(* CODESYS project tc3_mc3definitions.library
   TcLibraryId: Beckhoff Automation GmbH|Tc3_Mc3Definitions|3.2.38.0
   Company: Beckhoff Automation GmbH
   DefaultNamespace: Tc3_Mc3Definitions
   Version: 3.2.38.0
   Placeholder: Tc3_Mc3Definitions
   Title: Tc3_Mc3Definitions

Project tree, tasks and I/O mapping:
  Version/
    global variables Global_Version
  DUTs/
    Enums/
      data type MC_BUFFER_MODE
      data type MC_COMPENSATION_TYPE
      data type MC_DIRECTION
      data type MC_EXECUTION_MODE
      data type MC_SYNC_MODE
      data type MC_SYNC_STRATEGY
      data type MC_SYNC_DIRECTIONS
  GVLs/
    global variables GVL
*)

// DUTs/Enums/MC_BUFFER_MODE

(* Buffer mode between buffered commands. *)
	{attribute 'TcIecLibraryType'}
{attribute 'Namespace' := 'MC'}
TYPE MC_BUFFER_MODE : (mcAborting:=0, mcBuffered:=1, mcBlendingLow:=18, mcBlendingPrevious:=19, mcBlendingNext:=20, mcBlendingHigh:=21) UINT;
END_TYPE

// DUTs/Enums/MC_COMPENSATION_TYPE

(* Compensation type. *)
	{attribute 'TcIecLibraryType'}
{attribute 'Namespace' := 'MC'}
TYPE MC_COMPENSATION_TYPE : (mcTypeInvalidCompensation:=0, mcTypeGeoCompensation:=1) UINT;
END_TYPE

// DUTs/Enums/MC_DIRECTION

(* Defines the direction of the movement (e.g for an Modulo Axis). *)
	{attribute 'TcIecLibraryType'}
{attribute 'Namespace' := 'MC'}
TYPE MC_DIRECTION : (
	mcDirectionNonModulo:=0, 	(* Position is interpreted as absolute position. *)
	mcDirectionPositive:=1, 	(* Moves in positive direction. *)
	mcDirectionShortestWay:=2, 	(* The direction of movement depends on whether the positive direction of movement or the negative direction of movement is the shortest distance from the target position. *)
	mcDirectionNegative:=3	(* Moves in negative direction. *)
) UINT;
END_TYPE

// DUTs/Enums/MC_EXECUTION_MODE

(* Execution mode. *)
	{attribute 'TcIecLibraryType'}
{attribute 'Namespace' := 'MC'}
{attribute 'hide'}
TYPE MC_EXECUTION_MODE : (mcExecModeImmediately:=0, mcExecModeDelayed:=1, mcExecModeQueued:=2) UINT;
END_TYPE

// DUTs/Enums/MC_SYNC_MODE

(* Defines the direction of the synchronization position of modulo axes. *)
	{attribute 'TcIecLibraryType'}
{attribute 'Namespace' := 'MC'}
TYPE MC_SYNC_MODE : (
	mcSyncModeNonModulo:=0, 	(* SyncSlavePosition is interpreted as absolute position. *)
	mcSyncModePositive:=1, 	(* Synchronizes in positive direction. *)
	mcSyncModeNegative:=3	(* Synchronizes in negative direction. *)
) UINT;
END_TYPE

// DUTs/Enums/MC_SYNC_STRATEGY

(* Execution mode. *)
	{attribute 'TcIecLibraryType'}
{attribute 'Namespace' := 'MC'}
TYPE MC_SYNC_STRATEGY : (mcSyncStrategyLate:=1, mcSyncStrategySlow:=2, mcSyncStrategyEarly:=3) UINT;
END_TYPE

// DUTs/Enums/MC_SYNC_DIRECTIONS

(* Directions in which a slave is allowed to move during synchronizing phase. *)
	{attribute 'TcIecLibraryType'}
{attribute 'qualified_only'}
TYPE MC_SYNC_DIRECTIONS : (
		{attribute 'hide'}
Invalid:=0, 	(* Indicates invalid information, e.g. no connection or component not yet ready. *)
	Positive:=1, 	(* Movement is allowed only in positive direction while synchronizing. *)
	Negative:=2, 	(* Movement is allowed only in negative direction while synchronizing. *)
	Both:=3	(* Movement is allowed in any direction while synchronizing. *)
) UINT := Invalid;
END_TYPE

// Version/Global_Version
{attribute 'TcGenerated'}
// This function has been automatically generated from the project information.
VAR_GLOBAL CONSTANT
	{attribute 'const_non_replaced'}
	{attribute 'linkalways'}
	stLibVersion_Tc3_Mc3Definitions : ST_LibVersion := (iMajor := 3, iMinor := 2, iBuild := 38, iRevision := 0, sVersion := '3.2.38.0');
	{attribute 'const_non_replaced'}
	{attribute 'linkalways'}
	sLibraryId_Tc3_Mc3Definitions : String := 'Beckhoff Automation GmbH|Tc3_Mc3Definitions|3.2.38.0';
END_VAR

// GVLs/GVL

VAR_GLOBAL CONSTANT
		MC_DEFAULT	:	LREAL := 1E300;
		MC_IGNORE	:	LREAL := 1E301;
		MC_INVALID	:	LREAL := 1E302;
		MC_MAXIMUM	:	LREAL := 1E303;
	END_VAR
